FUNCTION_BLOCK PUBLIC CycleControl
VAR_IN_OUT
	
END_VAR
VAR_INPUT
END_VAR
VAR_OUTPUT
END_VAR
VAR
	bInitialize : BOOL := TRUE;
	bFirst: BOOL := TRUE;
	State : eCycleControlState := eCycleControlState.eUnknown;
	NextState : eCycleControlState := eCycleControlState.eUnknown;
	byCounter: BYTE :=1;
	StateTimer : TON;
	//fbPID: FB_CTRL_PID;
	CycleStopReq : BOOL := FALSE;
END_VAR

IF (bInitialize) THEN
	bInitialize := FALSE;
	// to add all initialization code here
END_IF


CASE State OF
eCycleControlState.eUnknown:
	IF (GVL_IO.MC_XStartPB AND GVL_IO.MC_XAirPressureOK AND GVL_IO.MC_NotEStopped) THEN // wait for start button when powered up or PLC program restarted
		NextState := eCycleControlState.eInit;	   
	END_IF
    StackLightRed();
	
	StateTimer(IN:=TRUE, PT:= T#10S); // give a message out every 10 seconds
	IF (StateTimer.Q) THEN
		Logging.fbEventMsg.SendEventMsg(MsgClass := TCEVENTCLASS_STATEINFO, EventID:= Logging.ID_CY_Unknown, SourceID:= Logging.SrcCyclePOU);
		StateTimer(IN:=FALSE);
	END_IF

eCycleControlState.eInit:
	IF (Stations.fbPrimeMover.WaitingForHomingTrigger) THEN  // checking to see if Magnemotion has completed software Path reset and HLC operational
		NextState := eCycleControlState.eWaitForHoming;
	END_IF
	StateTimer(IN:=TRUE, PT := T#250MS);
	IF (StateTimer.Q) THEN
		GVL_IO.MC_YStackLightRed := NOT GVL_IO.MC_YStackLightRed;
		GVL_IO.MC_YStackLightYellow := NOT GVL_IO.MC_YStackLightYellow;
		GVL_IO.MC_YStackLightGreen := NOT GVL_IO.MC_YStackLightGreen;
		StateTimer(IN:=FALSE);
	END_IF
	

eCycleControlState.eWaitForHoming:
	(*IF(Stations.fbPistonSta.Ready AND Stations.fbCapInsertSta.Ready AND Stations.fbGoodUnloadSta.Ready AND Stations.fbRejectSta.Ready) THEN
		NextState := eCycleControlState.eReady;
	END_IF *)
	StackLightYellow();
	IF(Stations.fbLoad1Sta.Ready AND
       Stations.fbVisionSta.Ready AND  
       Stations.fbPistonSta.Ready AND 
       Stations.fbCapInsertSta.Ready AND 
       //Stations.fbGoodUnloadSta.Ready AND
       Stations.fbGoodULSta_1.Ready AND
		Stations.fbGoodULSta_2.Ready AND
		Stations.fbGoodULSta_3.Ready AND
		Stations.fbGoodULSta_4.Ready AND     
		Stations.fbAutoBagger.Ready AND     
	   Stations.fbRejectSta.Ready  
       ) THEN
		NextState := eCycleControlState.eReady;
		StackLightGreen();
		Stations.fbPrimeMover.TriggerAction := TRUE; // Enable the Magnemotion controller bus propulsion
	END_IF

eCycleControlState.eReady:
	//IF (GVL_IO.MC_XStartPB) THEN //need to change this later
		NextState := eCycleControlState.eAutoRun;   //don't really need this start button again 			
	//END_IF	

eCycleControlState.eAutoRun:
	IF(bFirst) THEN
		FOR byCounter := 1 TO MM_CONST.MAX_VEHICLES BY 1 DO
			Stations.fbVehicleManager[byCounter].M_SetNextMoveParams(MM_CONST.REJECT_ULOAD_POS,2.0,2.0,MM_CONST.REJECT_ULOAD_STA);
			Stations.fbVehicleManager[byCounter].TriggerVehMov := TRUE;			
		END_FOR	
	END_IF
	// to do add logic here to handle cycle stop
	NextState := eCycleControlState.eStartStop ;

eCycleControlState.eStartStop:	
	IF( Stations.fbMMMonitor.IsMMJammed OR 
		Stations.fbLoad1Sta.IsFaulted() OR 
		NOT Stations.fbBurnOffSta.IsAtTemperature OR 
		Stations.fbVisionSta.IsFaulted() OR 
        Stations.fbPistonSta.IsFaulted() OR 
       Stations.fbCapInsertSta.IsFaulted() OR 
       //Stations.fbGoodUnloadSta.IsFaulted() OR
		Stations.fbGoodULSta_1.IsFaulted() OR
		Stations.fbGoodULSta_2.IsFaulted() OR
		Stations.fbGoodULSta_3.IsFaulted() OR
		Stations.fbGoodULSta_4.IsFaulted() OR
		Stations.fbAutoBagger.IsFaulted() OR		            
        Stations.fbRejectSta.IsFaulted()) 
       THEN 
			StackLightRed();
			GVL_IO.YU_YIMBADIsOK := FALSE;
	END_IF
	
    IF( NOT Stations.fbMMMonitor.IsMMJammed AND
		NOT Stations.fbLoad1Sta.IsFaulted() AND 
	    Stations.fbBurnOffSta.IsAtTemperature AND 
	    NOT Stations.fbVisionSta.IsFaulted() AND 
        NOT Stations.fbPistonSta.IsFaulted() AND 
        NOT Stations.fbCapInsertSta.IsFaulted() AND 
        //NOT Stations.fbGoodUnloadSta.IsFaulted() AND
        NOT Stations.fbGoodULSta_1.IsFaulted() AND
		NOT Stations.fbGoodULSta_2.IsFaulted() AND
		NOT Stations.fbGoodULSta_3.IsFaulted() AND
		NOT Stations.fbGoodULSta_4.IsFaulted() AND   
		NOT Stations.fbAutoBagger.IsFaulted() AND
        NOT Stations.fbRejectSta.IsFaulted()) 
    THEN 
			StackLightGreen(); 
			GVL_IO.YU_YIMBADIsOK := TRUE;
	END_IF
    
    IF (NOT GVL_IO.MC_XStopPB) THEN // hit the stop button
		CycleStopReq := TRUE;		
	END_IF
	
    IF (GVL_IO.MC_XStopPB AND GVL_IO.MC_XStartPB) THEN 
		CycleStopReq := FALSE;		
	END_IF
    
   IF (GVL_IO.MachineEStopped OR NOT GVL_IO.MC_XAirPressureOK ) THEN 
		NextState := eCycleControlState.eWaitForHomingAfterEStop;
		StackLightRed();
    END_IF
	
	IF CycleStopReq THEN
		StackLightYellow(); // we have a stop request
	END_IF
	
	
eCycleControlState.eWaitForHomingAfterEStop:

	IF (GVL_IO.MC_XAirPressureOK AND GVL_IO.MC_NotEStopped) THEN // wait for start button when powered up or PLC program restarted
		IF(Stations.fbPistonSta.Ready AND Stations.fbCapInsertSta.Ready
        //AND Stations.fbGoodUnloadSta.Ready
        AND Stations.fbGoodULSta_1.Ready
		AND Stations.fbGoodULSta_2.Ready
		AND Stations.fbGoodULSta_3.Ready
		AND Stations.fbGoodULSta_4.Ready 
        AND Stations.fbVisionSta.Ready ) THEN // Maybe add other stations here as well
			NextState := eCycleControlState.eStartStop;
			StackLightGreen();
		END_IF
		IF (GVL_IO.MC_XStopPB AND GVL_IO.MC_XStartPB) THEN
			CycleStopReq := FALSE;
			///Stations.fbMMSendMsg.M_CmdResumeMov(); // allow accepting commands for vehicle movement ?? Need to try this
		END_IF		
	END_IF
	
	
eCycleControlState.eError:	
//fbPID;

IF (GVL_IO.MC_XStartPB) THEN 
	GVL_IO.MC_YStackLightYellow := TRUE;
END_IF

END_CASE

IF (State <> NextState) THEN
	bFirst := TRUE;
	StateTimer(IN:=FALSE);
ELSE 
	bFirst := FALSE;	
END_IF

State := NextState;
Status.StationsState[MM_CONST.CYCLE_CONTROL_HMI_STATE] := State;
AssignStationStatusForHMI();
AssignErrorMessagetoHMI();

PROPERTY AllowPrimeMoverEnable : BOOL
GET
AllowPrimeMoverEnable := (State = eCycleControlState.eStartStop);
END_GET
END_PROPERTY

METHOD PUBLIC AssignErrorMessagetoHMI : BOOL
VAR_INPUT
END_VAR
IF (Stations.fbMMMonitor.IsMMJammed) THEN
	Status.ErrorMessage := Status.PrimeMoverStatusMsg;
ELSIF (Stations.fbLoad1Sta.IsFaulted()) THEN
	Status.ErrorMessage := Status.Load1StatusMsg;
ELSIF(Stations.fbVisionSta.IsFaulted()) THEN
	Status.ErrorMessage := Status.VisionStatusMsg;
ELSIF(Stations.fbPistonSta.IsFaulted()) THEN
	Status.ErrorMessage := Status.PistonStatusMsg;
ELSIF(Stations.fbCapInsertSta.IsFaulted()) THEN
	Status.ErrorMessage := Status.CapStatusMsg; 
//ELSIF(Stations.fbGoodUnloadSta.IsFaulted()) THEN
//	Status.ErrorMessage := Status.GoodULStatusMsg;    
ELSIF(Stations.fbGoodULSta_1.IsFaulted()) THEN
	Status.ErrorMessage := Status.GoodUL_1_StatusMsg;       
ELSIF(Stations.fbGoodULSta_2.IsFaulted()) THEN
	Status.ErrorMessage := Status.GoodUL_2_StatusMsg;
ELSIF(Stations.fbGoodULSta_3.IsFaulted()) THEN
	Status.ErrorMessage := Status.GoodUL_3_StatusMsg;
ELSIF(Stations.fbGoodULSta_4.IsFaulted()) THEN
	Status.ErrorMessage := Status.GoodUL_4_StatusMsg;
ELSIF(Stations.fbRejectSta.IsFaulted()) THEN
	Status.ErrorMessage := Status.RejectStatusMsg;
ELSIF(Stations.fbAutoBagger.IsFaulted()) THEN
	Status.ErrorMessage := Status.AutoBaggerStatusMsg;
ELSIF (Stations.fbLoad1Sta.IsLoadWaitingForYushin()) THEN
	Status.ErrorMessage := Status.Load1StatusMsg;	
ELSE
	Status.ErrorMessage := '';
END_IF
END_METHOD

METHOD PUBLIC AssignStationStatusForHMI : BOOL
VAR_INPUT
END_VAR
Status.StationsState[MM_CONST.CYCLE_CONTROL_HMI_STATE] := State;

CASE State OF 
	eCycleControlState.eUnknown, eCycleControlState.eError:
		Status.StationStauts[MM_CONST.CYCLE_CONTROL_HMI_STATE] := OverallStationStatus.eError;
    eCycleControlState.eInit,eCycleControlState.eWaitForHoming:
	    Status.StationStauts[MM_CONST.CYCLE_CONTROL_HMI_STATE] := OverallStationStatus.eHoming;
	eCycleControlState.eReady,eCycleControlState.eAutoRun,eCycleControlState.eStartStop:
	    IF (CycleStopReq) THEN
			Status.StationStauts[MM_CONST.CYCLE_CONTROL_HMI_STATE] := OverallStationStatus.eCycleStop;
        ELSE 
			Status.StationStauts[MM_CONST.CYCLE_CONTROL_HMI_STATE] := OverallStationStatus.eRunning;	
		END_IF
	    
	eCycleControlState.eWaitForHomingAfterEStop:
	    IF (GVL_IO.MC_XAirPressureOK AND GVL_IO.MC_NotEStopped) THEN
	         Status.StationStauts[MM_CONST.CYCLE_CONTROL_HMI_STATE] := OverallStationStatus.eHoming;
	    ELSE 
			Status.StationStauts[MM_CONST.CYCLE_CONTROL_HMI_STATE] := OverallStationStatus.eCycleStop;
		END_IF   
		
	ELSE;	
END_CASE
END_METHOD

METHOD PUBLIC ResetCycleControlState : BOOL
VAR_INPUT
END_VAR
State:= eCycleControlState.eUnknown;
NextState:= eCycleControlState.eUnknown;
CycleStopReq := FALSE;
END_METHOD

ACTION StackLightGreen:
GVL_IO.MC_YStackLightRed := FALSE;
GVL_IO.MC_YStackLightYellow := FALSE;
GVL_IO.MC_YStackLightGreen := TRUE;
END_ACTION

ACTION StackLightRed:
GVL_IO.MC_YStackLightRed := TRUE;
GVL_IO.MC_YStackLightYellow := FALSE;
GVL_IO.MC_YStackLightGreen := FALSE;
END_ACTION

ACTION StackLightYellow:
GVL_IO.MC_YStackLightRed := FALSE;
GVL_IO.MC_YStackLightYellow := TRUE;
GVL_IO.MC_YStackLightGreen := FALSE;
END_ACTION

PROPERTY PUBLIC StopRequested : BOOL
GET
StopRequested := CycleStopReq;
END_GET
SET // PUBLIC
CycleStopReq := StopRequested;
END_SET
END_PROPERTY

END_FUNCTION_BLOCK

(* stored: Version 1.1.0.1, ProductVersion 3.1.4022.6
   POU CycleControl: Id {58fdd113-ff46-484b-bc19-22c90b9891bd}, SpecialFunc None
   Property AllowPrimeMoverEnable: Id {5f4a2e5a-4a5f-43c2-a3f8-82087769331c}
   Get Get: Id {3196fff4-4ebc-4d02-b488-78f81e0b1cd5}
   Method AssignErrorMessagetoHMI: Id {d113c449-15a8-492f-9d46-0b24f9e78455}
   Method AssignStationStatusForHMI: Id {f190938e-20bb-4dae-83f5-35f6d694ca0e}
   Method ResetCycleControlState: Id {c33497ba-c3f3-4175-8736-bbfc84f27854}
   Action StackLightGreen: Id {a052c037-25db-44b5-8e42-fa7213d15246}
   Action StackLightRed: Id {8005133c-1b60-49d8-97ca-5d508d6d0a8f}
   Action StackLightYellow: Id {af2ca68d-32b0-4630-9a6e-83b4cea5d386}
   Property StopRequested: Id {5651dcfc-7127-4890-8cef-ea7d9c2f94ce}
   Get Get: Id {d3a7b526-c72d-49f4-8a3b-3c559b8c50a1}
   Set Set: Id {e777eac5-6337-412a-9d2a-a68f76ca98c2} *)
